PROGRAM MAIN
VAR
	parser : JsonParser;
    json : json_st := (name:='test', age:=23, car := 'supercar');
	fileMethod : ParserMethod := ParserMethod.WriteFile;
	runExecute : BOOL;
	hasError : BOOL;
	errorId : UDINT;
	filename : STRING := 'test.json';
END_VAR

parser(
	Execute:=runExecute, 
	File:= CONCAT('C:/testing/', filename), 
	ParseMethod:= TO_STRING(fileMethod),
	Content:= 'MAIN.json',
	Port := 851,
	HasError=> hasError, 
	ErrorId=> errorId);
	
IF runExecute THEN
	runExecute := FALSE;
END_IF

END_PROGRAM

(* stored: Version 1.1.0.1, ProductVersion 3.1.4024.4
   POU MAIN: Id {dbd58374-97a7-4ff4-9f5e-12b0f08c73ae}, SpecialFunc None *)
